Fanuc KAREL source: PROG_BACKUP.kl

PROGRAM T
%NOLOCKGROUP
VAR
 v0 : STRING[40]
 v1 : INTEGER
 v2 : INTEGER
 v3 : BOOLEAN
 v4 : INTEGER
BEGIN
 PROG_BACKUP(v0, v1, v2, v3, v4)
END T
